RESOURCE_TYPE _Core1
  (* Standard: 61499-2 *)
  (* Version 0.1, 2017-00-09, hpea485, UOA *)
  VAR_INPUT
    TxChanId : UDINT;
  END_VAR
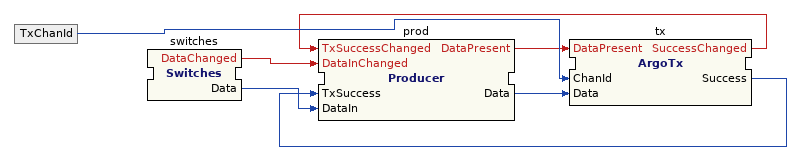
  FBS
    tx : ArgoTx;
    prod : Producer;
    switches : Switches;
  END_FBS
  EVENT_CONNECTIONS
    tx.SuccessChanged TO prod.TxSuccessChanged;
    prod.DataPresent TO tx.DataPresent;
    switches.DataChanged TO prod.DataInChanged;
  END_CONNECTIONS
  DATA_CONNECTIONS
    TxChanId TO tx.ChanId;
    tx.Success TO prod.TxSuccess;
    prod.Data TO tx.Data;
    switches.Data TO prod.DataIn;
  END_CONNECTIONS
END_RESOURCE_TYPE
